{attribute 'qualified_only'}
{attribute 'strict'}
TYPE E_Colors :
(
	red,
	orange,
	yellow,
	green,
	blue
);
END_TYPE

(* stored: Version 1.1.0.1, ProductVersion 3.1.4024.11
   DUT E_Colors: Id {a1f9771c-857e-4d96-915b-ed3836228790} *)
